// Mitsubishi GX Works2 project: 0605   PLC: Q00J
// 0605

PROGRAM MAIN
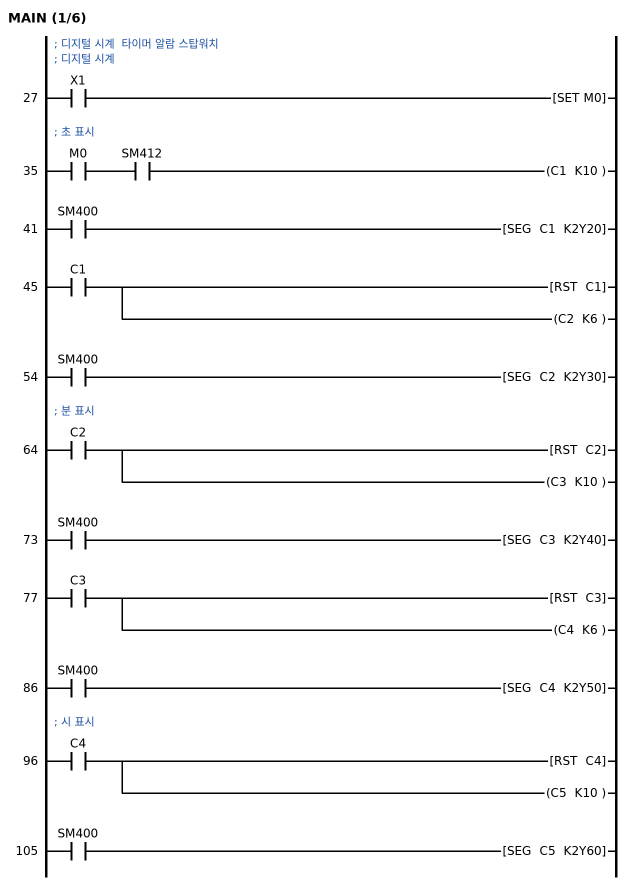
; 디지털 시계  타이머 알람 스탑워치
; 디지털 시계
27    LD      X1
      SET     M0
; 초 표시
35    LD      M0
      AND     SM412
      OUT     C1 K10
41    LD      SM400
      SEG     C1 K2Y20
45    LD      C1
      RST     C1
      OUT     C2 K6
54    LD      SM400
      SEG     C2 K2Y30
; 분 표시
64    LD      C2
      RST     C2
      OUT     C3 K10
73    LD      SM400
      SEG     C3 K2Y40
77    LD      C3
      RST     C3
      OUT     C4 K6
86    LD      SM400
      SEG     C4 K2Y50
; 시 표시
96    LD      C4
      RST     C4
      OUT     C5 K10
105   LD      SM400
      SEG     C5 K2Y60
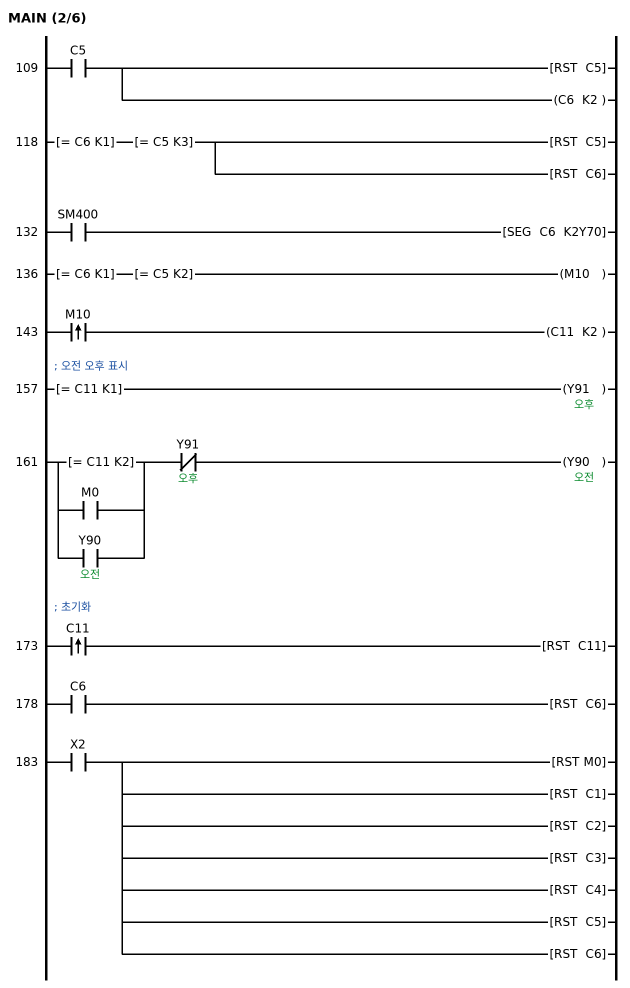
109   LD      C5
      RST     C5
      OUT     C6 K2
118   LD=     C6 K1
      AND=    C5 K3
      RST     C5
      RST     C6
132   LD      SM400
      SEG     C6 K2Y70
136   LD=     C6 K1
      AND=    C5 K2
      OUT     M10
143   LDP     M10
      OUT     C11 K2
; 오전 오후 표시
157   LD=     C11 K1
      OUT     Y91  ; 오후
161   LD=     C11 K2
      OR      M0
      OR      Y90  ; 오전
      ANI     Y91  ; 오후
      OUT     Y90  ; 오전
; 초기화
173   LDP     C11
      RST     C11
178   LD      C6
      RST     C6
183   LD      X2
      RST     M0
      RST     C1
      RST     C2
      RST     C3
      RST     C4
      RST     C5
      RST     C6
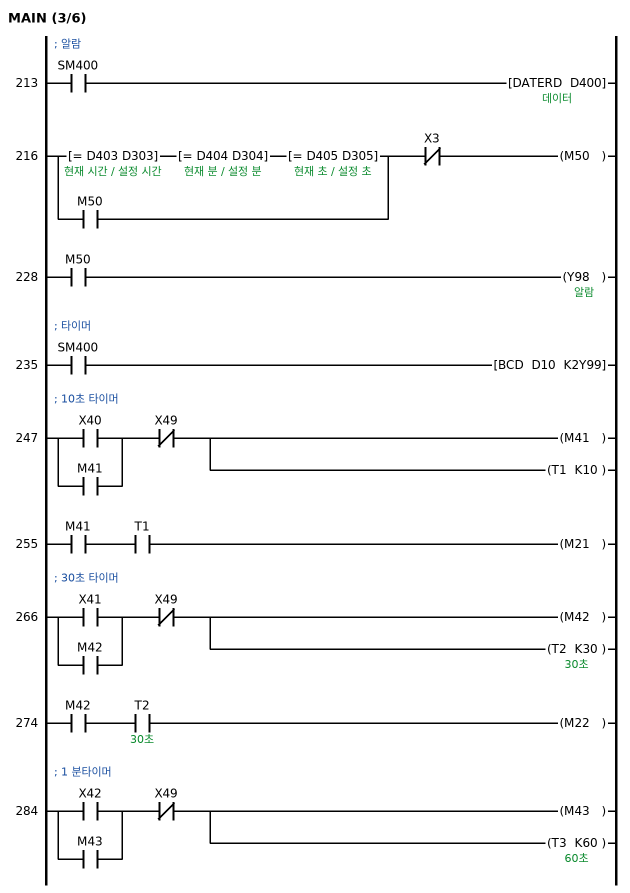
; 알람
213   LD      SM400
      DATERD  D400  ; 데이터
216   LD=     D403 D303  ; 현재 시간 / 설정 시간
      AND=    D404 D304  ; 현재 분 / 설정 분
      AND=    D405 D305  ; 현재 초 / 설정 초
      OR      M50
      ANI     X3
      OUT     M50
228   LD      M50
      OUT     Y98  ; 알람
; 타이머
235   LD      SM400
      BCD     D10 K2Y99
; 10초 타이머
247   LD      X40
      OR      M41
      ANI     X49
      OUT     M41
      OUT     T1 K10
255   LD      M41
      AND     T1
      OUT     M21
; 30초 타이머
266   LD      X41
      OR      M42
      ANI     X49
      OUT     M42
      OUT     T2 K30  ; 30초
274   LD      M42
      AND     T2  ; 30초
      OUT     M22
; 1 분타이머
284   LD      X42
      OR      M43
      ANI     X49
      OUT     M43
      OUT     T3 K60  ; 60초
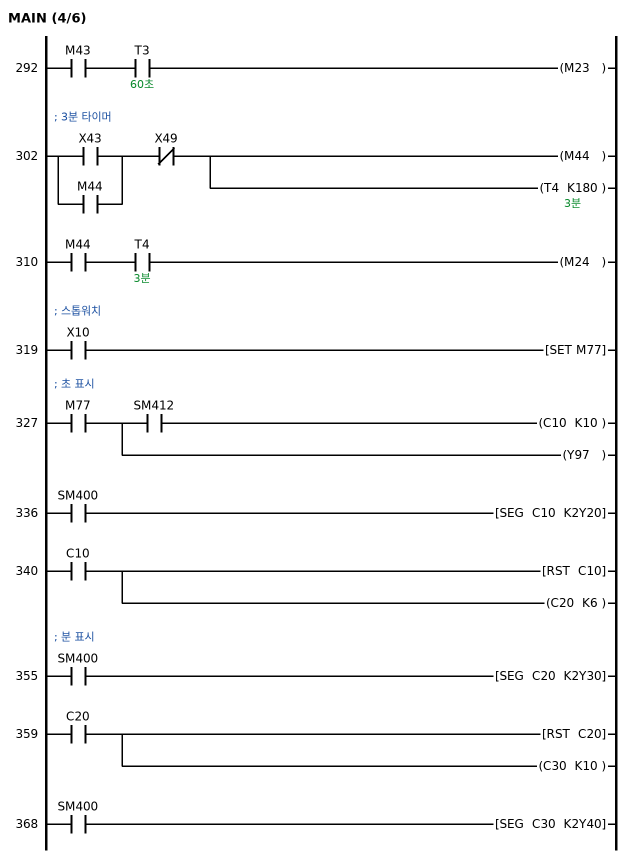
292   LD      M43
      AND     T3  ; 60초
      OUT     M23
; 3분 타이머
302   LD      X43
      OR      M44
      ANI     X49
      OUT     M44
      OUT     T4 K180  ; 3분
310   LD      M44
      AND     T4  ; 3분
      OUT     M24
; 스톱워치
319   LD      X10
      SET     M77
; 초 표시
327   LD      M77
      MPS
      AND     SM412
      OUT     C10 K10
      MPP
      OUT     Y97
336   LD      SM400
      SEG     C10 K2Y20
340   LD      C10
      RST     C10
      OUT     C20 K6
; 분 표시
355   LD      SM400
      SEG     C20 K2Y30
359   LD      C20
      RST     C20
      OUT     C30 K10
368   LD      SM400
      SEG     C30 K2Y40
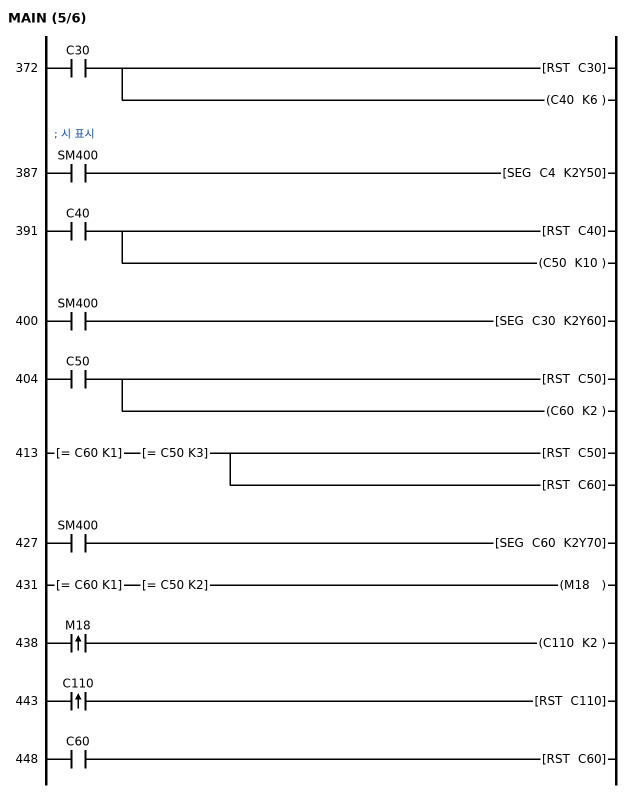
372   LD      C30
      RST     C30
      OUT     C40 K6
; 시 표시
387   LD      SM400
      SEG     C4 K2Y50
391   LD      C40
      RST     C40
      OUT     C50 K10
400   LD      SM400
      SEG     C30 K2Y60
404   LD      C50
      RST     C50
      OUT     C60 K2
413   LD=     C60 K1
      AND=    C50 K3
      RST     C50
      RST     C60
427   LD      SM400
      SEG     C60 K2Y70
431   LD=     C60 K1
      AND=    C50 K2
      OUT     M18
438   LDP     M18
      OUT     C110 K2
443   LDP     C110
      RST     C110
448   LD      C60
      RST     C60
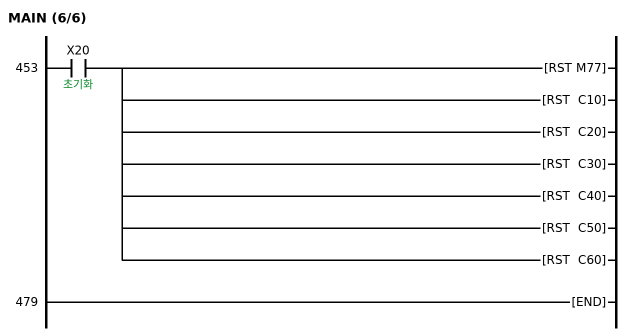
453   LD      X20  ; 초기화
      RST     M77
      RST     C10
      RST     C20
      RST     C30
      RST     C40
      RST     C50
      RST     C60
479   END
END_PROGRAM
